FUNCTION_BLOCK FB_AccelerationSensor IMPLEMENTS ITF_SubSystem
VAR_OUTPUT
	aAccelerationValues : ARRAY [0..2] OF REAL;
END_VAR
VAR
	//Local
	fbEL6001	: FB_SerialComRS232;
	fPacketRate : REAL := 0;
	bStartPacketCount : BOOL;
	
	fbTimer : TON;
	fbReset : TON;
	fbTrigger : R_TRIG;
	nCounter1 : UDINT;
	nCounter2 : UDINT;
	aPackets : ARRAY [0..9] OF UDINT;
	i : UDINT := 0;
	nSum : UDINT := 0;
	bTrigger : BOOL := FALSE;
	
	//ErrorBits
	bCommunicationError : BIT;
	bOutOfRange : BIT;
END_VAR
VAR CONSTANT
	fGravitationalAcceleration : REAL := 9.81;  					//in m/s^2
END_VAR

fbEL6001(stEL6001In:=AccelerationSensor.stEL6001In, stEL6001Out:=AccelerationSensor.stEL6001Out);

aAccelerationValues := fbEL6001.aAcceleration;

doPacketCount();

METHOD PRIVATE doCheckRange : BOOL
VAR_INPUT
	aValues : ARRAY [0..2] OF REAL;
	fMax : REAL;
END_VAR
IF ABS(aValues[0]) <= fMax AND ABS(aValues[1]) <= fMax AND ABS(aValues[2]) <= fMax THEN
	doCheckRange := TRUE;
ELSE
	doCheckRange := FALSE;
END_IF
END_METHOD

METHOD PRIVATE doPacketCount
VAR_INPUT
END_VAR
fbTimer(IN := bStartPacketCount, PT := T#1S);
fbTrigger(CLK := fbTimer.IN);

IF fbTrigger.Q THEN
	nCounter1 := fbEL6001.nReceiveCounter;
END_IF

IF fbTimer.Q THEN
	nCounter2 := fbEL6001.nReceiveCounter;
	aPackets[i] := nCounter2 - nCounter1;
	nSum := nSum + aPackets[i];
	i := i + 1;
	bTrigger := TRUE;
	bStartPacketCount := FALSE;
END_IF

IF i = 10 THEN
	bTrigger := FALSE;
	fPacketRate := (UDINT_TO_REAL(nSum) / UDINT_TO_REAL(i));
	i := 0;
	nSum := 0;
END_IF

fbReset(IN := bTrigger, PT := T#3S);
IF fbReset.Q THEN
	bStartPacketCount := TRUE;
	bTrigger := FALSE;
END_IF
END_METHOD

PROPERTY PUBLIC eCondition : SubLevelCondition
GET
IF nErrorID <> 0 THEN
	eCondition := SubLevelCondition.ERROR;
ELSE
	eCondition := SubLevelCondition.RUN;
END_IF
END_GET
END_PROPERTY

PROPERTY PUBLIC nErrorID : UDINT
GET
IF fbEL6001.eReceiveErrorID <> COMERROR_NOERROR THEN
	bCommunicationError := TRUE;
ELSE
	bCommunicationError := FALSE;
END_IF

bOutOfRange := NOT doCheckRange(aValues:=aAccelerationValues, fMax:=2*fGravitationalAcceleration);


nErrorID.0 := bCommunicationError;
nErrorID.1 := bOutOfRange;
END_GET
END_PROPERTY

END_FUNCTION_BLOCK

(* stored: Version 1.1.0.1, ProductVersion 3.1.4024.12
   POU FB_AccelerationSensor: Id {4efed543-46dd-452e-af75-10c16bcd4501}, SpecialFunc None
   Method doCheckRange: Id {94c692bc-79f2-4b46-aa0a-622a69a512a9}
   Method doPacketCount: Id {b6af9b40-4731-4ada-9b3a-8a6c4e7e8d93}
   Property eCondition: Id {fdc5f8c1-0576-4afe-aada-aa997b8b31b2}
   Get Get: Id {e176f809-39eb-4ab9-899c-e14f19656ceb}
   Property nErrorID: Id {3275ac9b-f517-42d6-8d31-0fe54b04eaa2}
   Get Get: Id {8e6a6a17-98f7-47e1-8f0f-c94b4219f6c5} *)
